(* IEC 61131-3 sources: CodesysTest/export/Function Blocks/Electric Solenoid/FB_ElectricSolenoid.pou/UpAsserted.prop, 1 file *)

(* ---- Get.pm.st ---- *)
(*#-#-#-#-#-#-#-#-#-#---Declaration---#-#-#-#-#-#-#-#-#-#-#-#-#*)

VAR
END_VAR
(*#-#-#-#-#-#-#-#-#-#---Implementation---#-#-#-#-#-#-#-#-#-#-#-#-#*)

UpAsserted := NOT actuateSolenoid;
